FUNCTION_BLOCK FB_Carro_DRC_LD
VAR_INPUT
    ManiobrasTotales: UINT := 2;
    TiempoEspera: TIME := T#2S;
END_VAR
VAR_OUTPUT
    ManiobrasPendientes: UINT;
    TiempoPendiente: TIME;
END_VAR
VAR
    // Estados futuros
    MarchaDerechaFuturo: BOOL;
    MarchaIzquierdaFuturo: BOOL;
    
    // Bloques funcionales
    FlancoPulsadorMarcha: R_TRIG;
    Intermitencia: FB_Blink;
    TemporizadorEspera: TON;
    ContadorManiobras: CTD;
    
    // Entradas
    i_PulsadorMarcha AT %I*: BOOL;
    i_FinalCarreraIzquierda AT %I*: BOOL := TRUE;
    i_FinalCarreraDerecha AT %I*: BOOL;
    
    // Salidas
    o_MarchaIzquierda AT %I*: BOOL;
    o_MarchaDerecha AT %I*: BOOL;
    o_LamparaMarcha AT %I*: BOOL;
END_VAR

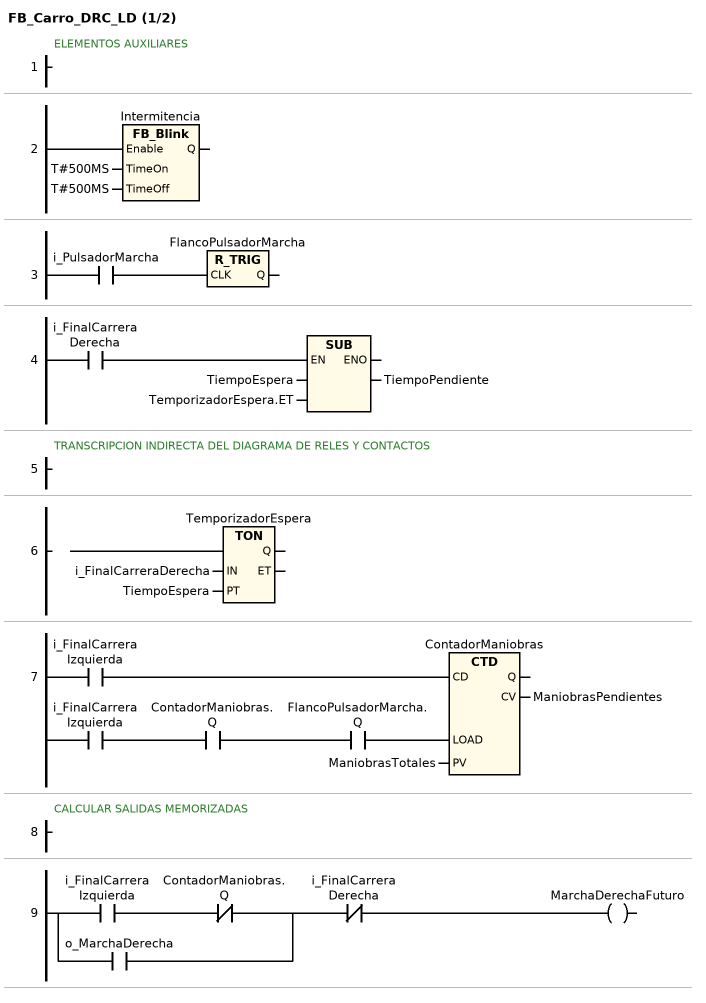
// NETWORK 1
// ELEMENTOS AUXILIARES

// NETWORK 2
Intermitencia(Enable := TRUE, TimeOn := T#500MS, TimeOff := T#500MS); // FB_Blink

// NETWORK 3
FlancoPulsadorMarcha(CLK := i_PulsadorMarcha); // R_TRIG

// NETWORK 4
IF i_FinalCarreraDerecha THEN TiempoPendiente := TiempoEspera - TemporizadorEspera.ET; END_IF

// NETWORK 5
// TRANSCRIPCION INDIRECTA DEL DIAGRAMA DE RELES Y CONTACTOS

// NETWORK 6
TemporizadorEspera(IN := i_FinalCarreraDerecha, PT := TiempoEspera); // TON

// NETWORK 7
ContadorManiobras(
    CD := i_FinalCarreraIzquierda,
    LOAD := i_FinalCarreraIzquierda AND ContadorManiobras.Q AND FlancoPulsadorMarcha.Q,
    PV := ManiobrasTotales,
    CV => ManiobrasPendientes); // CTD

// NETWORK 8
// CALCULAR SALIDAS MEMORIZADAS

// NETWORK 9
MarchaDerechaFuturo := (i_FinalCarreraIzquierda AND NOT ContadorManiobras.Q OR o_MarchaDerecha) AND NOT i_FinalCarreraDerecha;

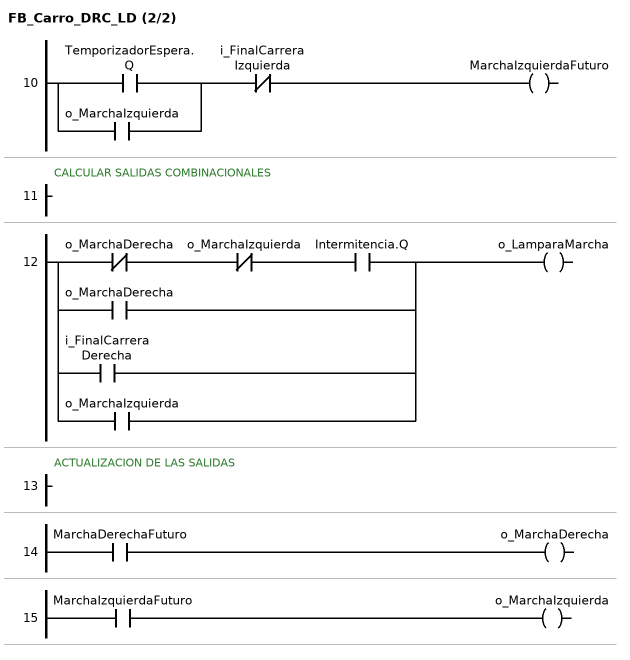
// NETWORK 10
MarchaIzquierdaFuturo := (TemporizadorEspera.Q OR o_MarchaIzquierda) AND NOT i_FinalCarreraIzquierda;

// NETWORK 11
// CALCULAR SALIDAS COMBINACIONALES

// NETWORK 12
o_LamparaMarcha := NOT o_MarchaDerecha AND NOT o_MarchaIzquierda AND Intermitencia.Q OR o_MarchaDerecha OR i_FinalCarreraDerecha OR o_MarchaIzquierda;

// NETWORK 13
// ACTUALIZACION DE LAS SALIDAS

// NETWORK 14
o_MarchaDerecha := MarchaDerechaFuturo;

// NETWORK 15
o_MarchaIzquierda := MarchaIzquierdaFuturo;

END_FUNCTION_BLOCK

(* stored: Version 1.1.0.1, ProductVersion 3.1.4024.16
   POU FB_Carro_DRC_LD: Id {95007db2-6afe-415c-a00b-f8f7958ae86c}, SpecialFunc None *)
